FUNCTION_BLOCK motor_starter
VAR_INPUT
	//Run Feedback from Motor Starter
	run_feedback : BOOL; 
	//Reset trigger for Runtime Maint
	runtime_maint_reset : BOOL;
	//Run Request from PLC Program
	run_request : BOOL;
	//Motor is faulted
	fault : BOOL;
	//Daily Reset from GENERAL POU
	daily_reset : BOOL;
END_VAR
VAR_OUTPUT
	//Tells the motor to start when true, stop when false
	run_command : BOOL;
	//Accumulated Runtime Hours Today
	runtime_today : REAL;
	//Accumulated Runtime Hours Today
	runtime_total : REAL;
	//Resettable Runtime for Maintenance purposes, Description is user adjustable
	runtime_maint : REAL;
	//Motor Status(Calculated) 0=Off, 1=Running, 2=Faulted
	status : INT;
END_VAR
VAR	
	//Runtime Timer Tags, 1 Minute Timer
	runtime_ton : TON;
	runtime_pt : TIME := T#1M;
	runtime_et : TIME;
	//Runtime Today Counter
	runtime_today_ctu : CTU;
	runtime_today_ctu_pv : WORD;
	runtime_today_ctu_cv : REAL;
	//Total Runtime Minute Counter
	runtime_total_minute_ctu : CTU;
	runtime_total_minute_ctu_reset : BOOL;
	runtime_total_minute_ctu_pv : WORD :=60;
	runtime_total_minute_ctu_cv : REAL;
	//Total Runtime Hour Counter
	runtime_total_hour_ctu : CTU;
	runtime_total_hour_ctu_reset : BOOL;
	runtime_total_hour_ctu_pv : WORD;
	//Maintenance Runtime Minute Counter
	runtime_maint_minute_ctu : CTU;
	runtime_maint_minute_cut_reset : BOOL;
	runtime_maint_minute_ctu_pv : WORD :=60;
	runtime_maint_minute_ctu_cv : REAL;
	//Maintenance Runtime Hour Counter
	runtime_maint_hour_ctu : CTU;
	runtime_maint_hour_ctu_pv : WORD;
END_VAR
VAR // added by the converter: edge detectors and wires of the graphical bodies
    _w1, _w2, _w3 : BOOL;
END_VAR

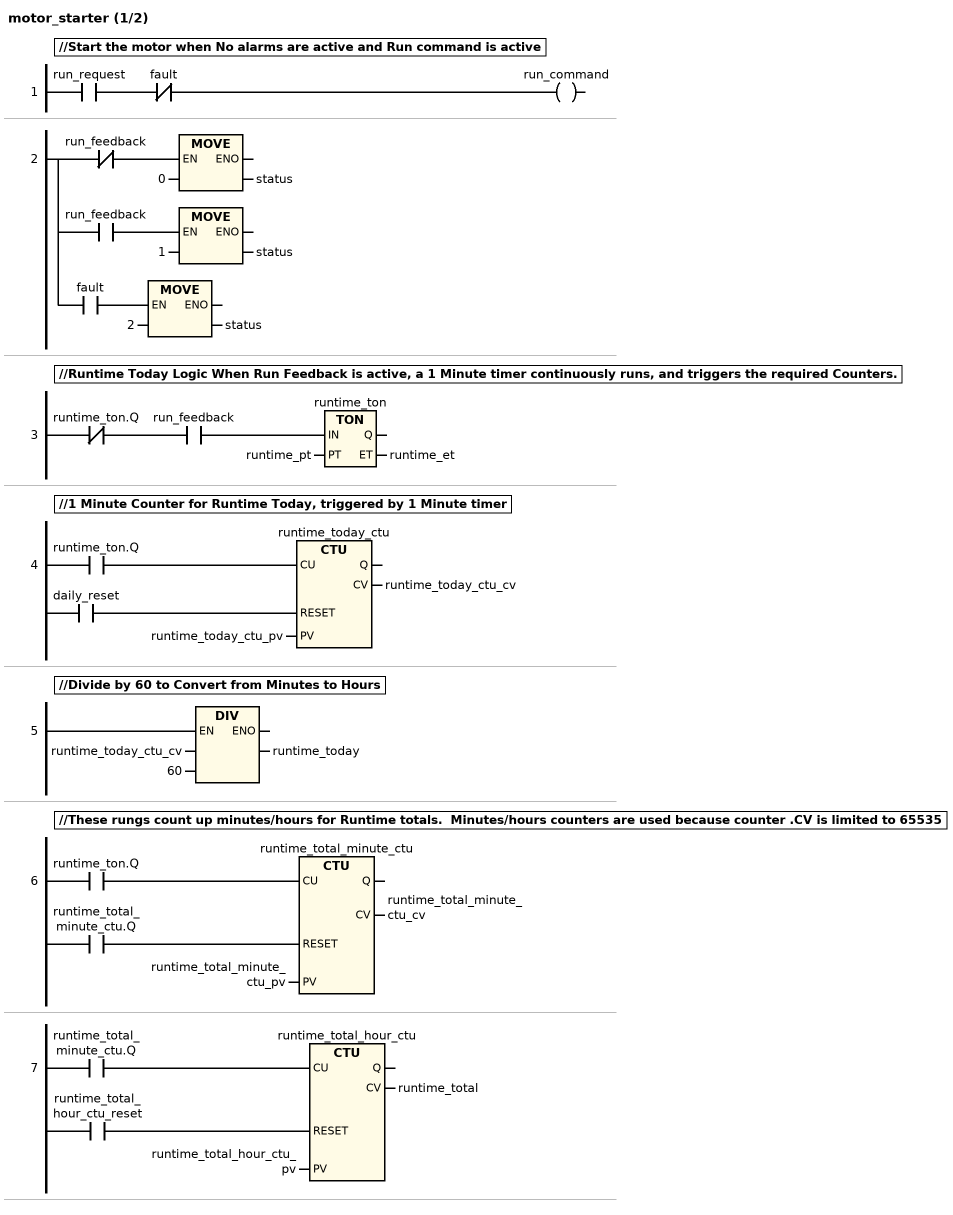
// NETWORK 1
// label: //Start the motor when No alarms are active and Run command is active
run_command := run_request AND NOT fault;

// NETWORK 2
_w1 := NOT run_feedback;
IF _w1 THEN status := 0; END_IF
_w2 := run_feedback;
IF _w2 THEN status := 1; END_IF
_w3 := fault;
IF _w3 THEN status := 2; END_IF
(* _w1 OR _w2 OR _w3; result not used *)

// NETWORK 3
// label: //Runtime Today Logic When Run Feedback is active, a 1 Minute timer continuously runs, and triggers the required Counters.
runtime_ton(IN := NOT runtime_ton.Q AND run_feedback, PT := runtime_pt, ET => runtime_et); // TON

// NETWORK 4
// label: //1 Minute Counter for Runtime Today, triggered by 1 Minute timer
runtime_today_ctu(
    CU := runtime_ton.Q,
    RESET := daily_reset,
    PV := runtime_today_ctu_pv,
    CV => runtime_today_ctu_cv); // CTU

// NETWORK 5
// label: //Divide by 60 to Convert from Minutes to Hours
runtime_today := runtime_today_ctu_cv / 60;

// NETWORK 6
// label: //These rungs count up minutes/hours for Runtime totals.  Minutes/hours counters are used because counter .CV is limited to 65535
runtime_total_minute_ctu(
    CU := runtime_ton.Q,
    RESET := runtime_total_minute_ctu.Q,
    PV := runtime_total_minute_ctu_pv,
    CV => runtime_total_minute_ctu_cv); // CTU

// NETWORK 7
runtime_total_hour_ctu(
    CU := runtime_total_minute_ctu.Q,
    RESET := runtime_total_hour_ctu_reset,
    PV := runtime_total_hour_ctu_pv,
    CV => runtime_total); // CTU

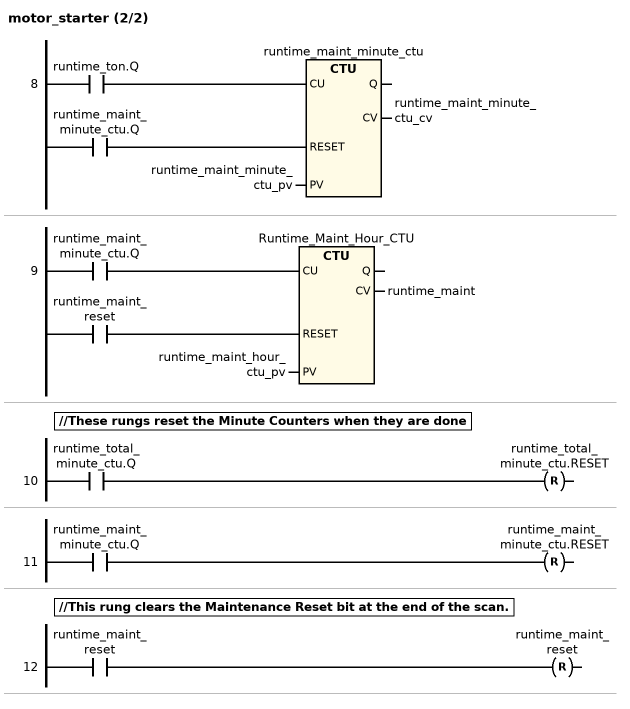
// NETWORK 8
runtime_maint_minute_ctu(
    CU := runtime_ton.Q,
    RESET := runtime_maint_minute_ctu.Q,
    PV := runtime_maint_minute_ctu_pv,
    CV => runtime_maint_minute_ctu_cv); // CTU

// NETWORK 9
Runtime_Maint_Hour_CTU(
    CU := runtime_maint_minute_ctu.Q,
    RESET := runtime_maint_reset,
    PV := runtime_maint_hour_ctu_pv,
    CV => runtime_maint); // CTU

// NETWORK 10
// label: //These rungs reset the Minute Counters when they are done
runtime_total_minute_ctu.RESET R= runtime_total_minute_ctu.Q;

// NETWORK 11
runtime_maint_minute_ctu.RESET R= runtime_maint_minute_ctu.Q;

// NETWORK 12
// label: //This rung clears the Maintenance Reset bit at the end of the scan.
runtime_maint_reset R= runtime_maint_reset;

END_FUNCTION_BLOCK

(* stored: Version 1.1.0.1, ProductVersion 3.1.4024.12
   POU motor_starter: Id {0dc68c89-7bb5-4fd3-a863-492b30a062fa}, SpecialFunc None *)
